// SIMATIC S7-200 project (STEP 7-Micro/WIN), CPU 224 CN REL 02.01

SYMBOL_TABLE 用户定义2
A灯电流             AIW0
B灯电流             AIW2
C灯电流             AIW4
外部机器速度           AIW6
A灯温度             AIW8
B灯温度             AIW10
C灯温度             AIW12
冷水机温度            AIW14
调光变频器频率          AQW0
风机变频器频率          AQW2
急停               I0.0
水流开关             I0.1
变压器A超温           I0.2
变压器B超温           I0.3
变压器C超温           I0.4
A灯限位             I0.5
B灯限位             I0.6
C灯限位             I0.7
A灯快门开启信号         I1.0
B灯快门开启信号         I1.1
C灯快门开启信号         I1.2
长车信号             I1.3
合压信号             I1.4
低水位检测            I1.5
制冷故障             I2.0
风机变频故障           I2.1
冷却系统启动           Q0.0
风机变频启动           Q0.1
A灯启动             Q0.2
B灯启动             Q0.3
C灯启动             Q0.4
A灯开启75           Q0.5
A灯开启100          Q0.6
B灯开启75           Q0.7
B灯开启100          Q1.0
C灯开启75           Q1.1
C灯开启100          Q2.0
A灯快门开启           Q2.1
B灯快门开启           Q2.2
C灯快门开启           Q2.3
报警输出             Q2.4
风机变频复位           Q2.5
风机选择             Q2.6
END_SYMBOL_TABLE

ORGANIZATION_BLOCK 主程序:OB1
TITLE=应用于印刷厂UV固化生产线的PLC控制系统。负责管理照明系统（A灯启动、B灯启动、C灯启动）、冷却系统（冷却系统启动）和通风系统（风机变频启动），确保油墨固化过程在安全、高效的条件下进行。
// 系统通过水流开关和低水位检测监测水况，并在水流正常且水位充足时激活冷却系统启动，为生产线提供稳定的散热支持。
// 冷却系统启动时必须确保水流正常。若冷水机温度超过设定值，系统暂停冷却系统启动并置位报警输出。水流开关检测到异常时，触发报警输出以提示操作员。操作员通过报警复位手动清除报警输出状态，报警复位后应确保报警条件已解除。
// 生产线上的A灯启动、B灯启动、C灯启动分别控制三组UV灯，用于固化不同区域的印刷油墨。这些灯的运行依赖于A灯温度、B灯温度、C灯温度的实时监测，只有在温度低于安全阈值、冷却系统启动和风机变频启动正常运行，且变压器A超温、变压器B超温、变压器C超温未触发时，灯才能开启。A灯启动时，A灯快门保持关闭状态。灯的亮度通过A灯开启75、A灯开启100等输出根据外部机器速度动态调节，确保固化效果与生产节奏匹配。此外，A灯快门开启、B灯快门开启、C灯快门开启在合压信号和长车信号确认生产线处于特定状态时打开，快门开启应在灯启动后特定时间触发。计时器阈值根据生产需求初始化为固定值，存储在系统中。
// 风机变频启动通过风机选择切换模式并在无风机变频故障时启动，为生产线提供通风散热。系统还配备保护机制，例如当A灯限位、B灯限位、C灯限位触发时，激活报警输出并关闭相关灯。急停按钮允许操作员随时中断冷却系统启动等关键输出，确保紧急情况下安全。在实际运行中，系统通过数据处理子程序采集A灯电流、B灯电流、C灯电流和温度数据，调整调光变频器频率和风机变频器频率，优化能耗与性能。生产线运行时间由系统累计记录，并与设定值比较以控制设备状态。当生产线运行时间达到或超过设定值时，停止所有灯。
// 
BEGIN
Network 1 // 网络标题
// 网络注释
LD     SM0.1
R      冷却系统启动:Q0.0, 100
R      M0.0, 100
R      M10.0, 100
R      V1000.0, 26
R      V1003.3, 100
S      M20.0, 1
R      V2700.0, 8
Network 2
LD     M20.0
TON    T45, +300
Network 3
LD     水流开关:I0.1
EU
R      M20.0, 1
Network 4
LD     T45
AN     水流开关:I0.1
S      报警输出:Q2.4, 1
S      V1000.5, 1
Network 5
LD     T45
AN     低水位检测:I1.5
R      A灯启动:Q0.2, 12
S      V1000.6, 1
S      报警输出:Q2.4, 1
R      冷却系统启动:Q0.0, 1
S      M13.7, 1
Network 7
LD     T45
R      M20.0, 1
Network 9
LD     SM0.0
CALL   运行:SBR0
Network 10
LD     SM0.0
CALL   报警:SBR1
Network 11
LD     SM0.0
CALL   数据处理:SBR2
Network 12
LDN    急停:I0.0
R      冷却系统启动:Q0.0, 100
R      M0.0, 100
END_ORGANIZATION_BLOCK

SUBROUTINE_BLOCK 运行:SBR0
TITLE=子程序注释
BEGIN
Network 2
LD     M1.1
EU
AN     制冷故障:I2.0
AW<=   VW806, VW206
A      低水位检测:I1.5
S      冷却系统启动:Q0.0, 1
Network 3
LD     M1.1
ED
R      冷却系统启动:Q0.0, 1
Network 4
LD     M6.0
EU
S      风机选择:Q2.6, 1
Network 5
LD     风机选择:Q2.6
ED
R      M6.0, 1
R      A灯启动:Q0.2, 18
Network 6
LD     冷却系统启动:Q0.0
ED
R      M0.3, 7
R      A灯启动:Q0.2, 18
R      M1.3, 12
Network 7
LD     风机变频启动:Q0.1
ED
R      A灯启动:Q0.2, 18
Network 9
LD     M6.0
ED
R      风机选择:Q2.6, 1
Network 10
LD     M1.2
EU
A      风机选择:Q2.6
AN     风机变频故障:I2.1
S      风机变频启动:Q0.1, 1
Network 11
LD     M1.2
ED
R      风机变频启动:Q0.1, 1
Network 12
LD     M0.3
EU
A      冷却系统启动:Q0.0
A      风机变频启动:Q0.1
AW<=   VW800, VW200
AN     A灯限位:I0.5
AN     V1001.0
A      变压器A超温:I0.2
AN     V1001.1
S      A灯启动:Q0.2, 1
Network 13
LDW>=  VW418, VW2500
A      A灯启动:Q0.2
A      T40
S      A灯开启75:Q0.5, 1
Network 14
LDW<   VW418, VW2600
R      A灯开启75:Q0.5, 1
Network 15
LDW>=  VW418, VW2502
A      A灯启动:Q0.2
A      T40
S      A灯开启100:Q0.6, 1
Network 16
LDW<   VW418, VW2602
R      A灯开启100:Q0.6, 1
Network 17
LD     M0.5
EU
A      冷却系统启动:Q0.0
A      风机变频启动:Q0.1
AW<=   VW802, VW202
AN     B灯限位:I0.6
A      变压器B超温:I0.3
AN     V1001.2
AN     V1001.3
S      B灯启动:Q0.3, 1
Network 18
LDW>=  VW418, VW2504
A      B灯启动:Q0.3
A      T46
S      B灯开启75:Q0.7, 1
Network 19
LDW<   VW418, VW2604
R      B灯开启75:Q0.7, 1
Network 20
LDW>=  VW418, VW2506
A      B灯启动:Q0.3
A      T46
S      B灯开启100:Q1.0, 1
Network 21
LDW<   VW418, VW2606
R      B灯开启100:Q1.0, 1
Network 22
LD     M0.7
EU
A      冷却系统启动:Q0.0
A      风机变频启动:Q0.1
AW<=   VW804, VW204
AN     C灯限位:I0.7
A      变压器C超温:I0.4
AN     V1001.4
AN     V1001.5
S      C灯启动:Q0.4, 1
Network 23
LDW>=  VW418, VW2508
A      C灯启动:Q0.4
A      T47
S      C灯开启75:Q1.1, 1
Network 24
LDW<   VW418, VW2608
R      C灯开启75:Q1.1, 1
Network 25
LDW>=  VW418, VW2510
A      C灯启动:Q0.4
A      T47
S      C灯开启100:Q2.0, 1
Network 26
LDW<   VW418, VW2610
R      C灯开启100:Q2.0, 1
Network 27
LD     M0.4
EU
R      A灯启动:Q0.2, 1
R      A灯开启75:Q0.5, 2
Network 28
LD     M0.6
EU
R      B灯启动:Q0.3, 1
R      B灯开启75:Q0.7, 2
Network 29
LD     M1.0
EU
R      C灯启动:Q0.4, 1
R      C灯开启75:Q1.1, 2
Network 30
LD     合压信号:I1.4
EU
A      长车信号:I1.3
LPS
A      A灯启动:Q0.2
A      T40
AW>=   VW418, VW3000
S      A灯快门开启:Q2.1, 1
LRD
A      B灯启动:Q0.3
A      T46
AW>=   VW418, VW3000
S      B灯快门开启:Q2.2, 1
LPP
A      C灯启动:Q0.4
A      T47
AW>=   VW418, VW3000
S      C灯快门开启:Q2.3, 1
Network 31
LD     T40
EU
A      合压信号:I1.4
A      长车信号:I1.3
A      A灯启动:Q0.2
AW>=   VW418, VW3000
S      A灯快门开启:Q2.1, 1
Network 32
LD     T46
EU
A      合压信号:I1.4
A      长车信号:I1.3
A      B灯启动:Q0.3
AW>=   VW418, VW3000
S      B灯快门开启:Q2.2, 1
Network 33
LD     T47
EU
A      合压信号:I1.4
A      长车信号:I1.3
A      C灯启动:Q0.4
AW>=   VW418, VW3000
S      C灯快门开启:Q2.3, 1
Network 34
LDW>=  VW418, VW3000
EU
A      合压信号:I1.4
A      长车信号:I1.3
LPS
A      A灯启动:Q0.2
A      T40
S      A灯快门开启:Q2.1, 1
LRD
A      B灯启动:Q0.3
A      T46
S      B灯快门开启:Q2.2, 1
LPP
A      C灯启动:Q0.4
A      T47
S      C灯快门开启:Q2.3, 1
Network 35
LDW<   VW418, VW3000
EU
LD     A灯快门开启:Q2.1
O      B灯快门开启:Q2.2
O      C灯快门开启:Q2.3
ALD
R      A灯快门开启:Q2.1, 1
R      B灯快门开启:Q2.2, 1
R      C灯快门开启:Q2.3, 1
Network 46
LD     A灯启动:Q0.2
ED
R      A灯快门开启:Q2.1, 1
Network 47
LD     B灯启动:Q0.3
ED
R      B灯快门开启:Q2.2, 1
Network 48
LD     C灯启动:Q0.4
ED
R      C灯快门开启:Q2.3, 1
Network 51
LD     合压信号:I1.4
ED
A      长车信号:I1.3
LD     A灯快门开启:Q2.1
O      B灯快门开启:Q2.2
O      C灯快门开启:Q2.3
ALD
S      M5.0, 2
Network 52
LD     合压信号:I1.4
EU
A      M5.0
R      M5.0, 1
Network 53
LD     M5.0
TON    T38, VW150
Network 54
LD     T38
EU
R      A灯快门开启:Q2.1, 3
R      M5.0, 1
Network 55
LDN    合压信号:I1.4
A      长车信号:I1.3
LD     A灯启动:Q0.2
O      B灯启动:Q0.3
O      C灯启动:Q0.4
ALD
S      M9.0, 1
Network 56
LDN    合压信号:I1.4
ED
A      长车信号:I1.3
R      M9.0, 1
Network 57
LD     长车信号:I1.3
ED
R      M9.0, 1
Network 58
LD     M9.0
EU
BITIM  VD350
Network 59
LD     M9.0
CITIM  VD350, VD354
Network 60
LD     M9.0
ED
MOVD   +0, VD350
MOVD   +0, VD354
Network 61
LDD>=  VD354, VD304
EU
R      A灯启动:Q0.2, 18
S      报警输出:Q2.4, 1
S      V1000.2, 1
S      M14.1, 1
Network 62
LD     A灯启动:Q0.2
TON    T40, VW2002
Network 63
LD     B灯启动:Q0.3
TON    T46, VW2002
Network 64
LD     C灯启动:Q0.4
TON    T47, VW2002
Network 65
LD     T40
O      T46
O      T47
EU
S      V1003.2, 1
Network 66
LDN    A灯启动:Q0.2
AN     B灯启动:Q0.3
AN     C灯启动:Q0.4
R      V1003.2, 1
Network 69
LD     M7.0
EU
AN     A灯启动:Q0.2
AN     B灯启动:Q0.3
AN     C灯启动:Q0.4
S      A灯快门开启:Q2.1, 1
Network 70
LD     M7.0
ED
AN     A灯启动:Q0.2
AN     B灯启动:Q0.3
AN     C灯启动:Q0.4
R      A灯快门开启:Q2.1, 1
Network 71
LD     M7.1
EU
AN     A灯启动:Q0.2
AN     B灯启动:Q0.3
AN     C灯启动:Q0.4
S      B灯快门开启:Q2.2, 1
Network 72
LD     M7.1
ED
AN     A灯启动:Q0.2
AN     B灯启动:Q0.3
AN     C灯启动:Q0.4
R      B灯快门开启:Q2.2, 1
Network 73
LD     M7.2
EU
AN     A灯启动:Q0.2
AN     B灯启动:Q0.3
AN     C灯启动:Q0.4
S      C灯快门开启:Q2.3, 1
Network 74
LD     M7.2
ED
AN     A灯启动:Q0.2
AN     B灯启动:Q0.3
AN     C灯启动:Q0.4
R      C灯快门开启:Q2.3, 1
Network 75
LDN    A灯开启75:Q0.5
AN     A灯开启100:Q0.6
A      A灯启动:Q0.2
S      Q1.5, 1
Network 76
LD     A灯开启75:Q0.5
O      A灯开启100:Q0.6
R      Q1.5, 1
Network 77
LD     A灯启动:Q0.2
ED
R      Q1.5, 1
R      A灯开启75:Q0.5, 2
Network 78
LDN    B灯开启75:Q0.7
AN     B灯开启100:Q1.0
A      B灯启动:Q0.3
S      Q1.6, 1
Network 79
LD     B灯开启75:Q0.7
O      B灯开启100:Q1.0
R      Q1.6, 1
Network 80
LD     B灯启动:Q0.3
ED
R      Q1.6, 1
R      B灯开启75:Q0.7, 2
Network 82
LDN    C灯开启75:Q1.1
AN     C灯开启100:Q2.0
A      C灯启动:Q0.4
S      Q1.7, 1
Network 83
LD     C灯开启75:Q1.1
O      C灯开启100:Q2.0
R      Q1.7, 1
Network 84
LD     C灯启动:Q0.4
ED
R      Q1.7, 1
R      C灯开启75:Q1.1, 1
R      C灯开启100:Q2.0, 1
END_SUBROUTINE_BLOCK

SUBROUTINE_BLOCK 报警:SBR1
TITLE=
BEGIN
Network 1
LD     M10.0
R      报警输出:Q2.4, 1
R      V1000.3, 100
R      V1000.0, 26
R      M17.0, 4
R      M9.0, 1
Network 2
LDW>   VW520, +120
EU
A      A灯启动:Q0.2
A      T49
S      V2700.0, 1
Network 3
LD     T49
EU
A      A灯启动:Q0.2
AW>    VW520, +120
S      V2700.0, 1
Network 4
LD     V2700.0
TON    T120, 20
Network 5
LD     T120
EU
AW>    VW520, +120
S      V1001.0, 1
S      报警输出:Q2.4, 1
R      A灯启动:Q0.2, 1
R      A灯开启75:Q0.5, 2
R      V2700.0, 1
Network 6
LD     T120
EU
R      V2700.0, 1
Network 7
LDW<   VW520, 40
EU
A      A灯启动:Q0.2
A      T49
S      V2700.1, 1
Network 8
LD     T49
EU
A      A灯启动:Q0.2
AW<    VW520, 40
S      V2700.1, 1
Network 9
LD     V2700.1
TON    T121, 20
Network 10
LD     T121
EU
AW<    VW520, 40
S      V1001.1, 1
S      报警输出:Q2.4, 1
R      A灯启动:Q0.2, 1
R      A灯开启75:Q0.5, 2
R      V2700.1, 1
Network 11
LD     T121
EU
R      V2700.1, 1
Network 14
LD     A灯启动:Q0.2
TON    T49, +300
Network 17
LDW>   VW620, +120
EU
A      B灯启动:Q0.3
A      T50
S      V2700.2, 1
Network 18
LD     T50
EU
AW>    VW620, +120
S      V2700.2, 1
Network 19
LD     V2700.2
TON    T122, 20
Network 20
LD     T122
EU
AW>    VW620, +120
S      V1001.2, 1
S      报警输出:Q2.4, 1
R      B灯启动:Q0.3, 1
R      B灯开启75:Q0.7, 2
R      V2700.2, 1
Network 21
LD     T122
EU
R      V2700.2, 1
Network 23
LD     B灯启动:Q0.3
TON    T50, +300
Network 25
LDW<   VW620, 40
EU
A      B灯启动:Q0.3
A      T50
S      V2700.3, 1
Network 26
LD     T50
EU
A      B灯启动:Q0.3
AW<    VW620, 40
S      V2700.3, 1
Network 27
LD     V2700.3
TON    T123, 20
Network 28
LD     T123
EU
AW<    VW620, 40
S      V1001.3, 1
S      报警输出:Q2.4, 1
R      B灯启动:Q0.3, 1
R      B灯开启75:Q0.7, 2
R      V2700.3, 1
Network 29
LD     T123
EU
R      V2700.3, 1
Network 32
LDW>   VW720, +120
EU
A      C灯启动:Q0.4
A      T51
S      V2700.4, 1
Network 33
LD     T51
EU
A      C灯启动:Q0.4
AW>    VW720, +120
S      V2700.4, 1
Network 34
LD     V2700.4
TON    T124, 20
Network 35
LD     T124
EU
AW>    VW720, +120
S      V1001.4, 1
S      报警输出:Q2.4, 1
R      C灯启动:Q0.4, 1
R      C灯开启75:Q1.1, 2
R      V2700.4, 1
Network 36
LD     T124
EU
R      V2700.4, 1
Network 37
LDW<   VW720, 40
EU
A      C灯启动:Q0.4
A      T51
S      V2700.5, 1
Network 38
LD     T51
EU
A      C灯启动:Q0.4
AW<    VW720, 40
S      V2700.5, 1
Network 39
LD     V2700.5
TON    T125, 20
Network 40
LD     T125
EU
AW<    VW720, 40
S      V1001.5, 1
S      报警输出:Q2.4, 1
R      C灯启动:Q0.4, 1
R      C灯开启75:Q1.1, 2
R      V2700.5, 1
Network 41
LD     T125
EU
R      V2700.5, 1
Network 44
LD     C灯启动:Q0.4
TON    T51, +300
Network 46
LDW>   VW800, VW200
EU
S      M17.0, 1
Network 47
LD     M17.0
TON    T102, 60
Network 48
LD     T102
EU
AW>    VW800, VW200
S      V1001.6, 1
R      A灯启动:Q0.2, 1
S      报警输出:Q2.4, 1
R      A灯开启75:Q0.5, 2
R      M17.0, 1
Network 49
LD     T102
EU
R      M17.0, 1
Network 51
LDW>   VW802, VW202
EU
S      M17.1, 1
Network 52
LD     M17.1
TON    T103, +60
Network 53
LD     T103
EU
AW>    VW802, VW202
S      V1001.7, 1
R      B灯启动:Q0.3, 1
S      报警输出:Q2.4, 1
R      B灯开启75:Q0.7, 2
R      M17.1, 1
Network 54
LD     T103
EU
R      M17.1, 1
Network 57
LDW>   VW804, VW204
EU
S      M17.2, 1
Network 58
LD     M17.2
TON    T104, +60
Network 59
LD     T104
EU
AW>    VW804, VW204
S      V1000.0, 1
R      C灯启动:Q0.4, 1
S      报警输出:Q2.4, 1
R      C灯开启75:Q1.1, 2
R      M17.2, 1
Network 60
LD     T104
EU
R      M17.2, 1
Network 64
LDW>   VW806, VW206
EU
AN     M20.0
S      M17.3, 1
Network 65
LD     M17.3
TON    T105, +60
Network 66
LD     T105
EU
AW>    VW806, VW206
S      V1000.1, 1
R      冷却系统启动:Q0.0, 1
S      报警输出:Q2.4, 1
R      风机变频复位:Q2.5, 2
R      A灯启动:Q0.2, 20
S      M13.0, 1
R      M17.3, 1
Network 67
LD     T105
EU
R      M17.3, 1
Network 70
LD     制冷故障:I2.0
EU
S      M13.1, 1
Network 71
LD     M13.1
TON    T60, +50
Network 72
LD     T60
EU
A      制冷故障:I2.0
R      冷却系统启动:Q0.0, 1
R      A灯启动:Q0.2, 20
R      风机变频复位:Q2.5, 2
S      V1000.3, 1
S      报警输出:Q2.4, 1
R      M13.1, 1
Network 73
LD     T60
AN     制冷故障:I2.0
R      M13.1, 1
Network 75
LDN    变压器A超温:I0.2
EU
R      A灯启动:Q0.2, 1
S      报警输出:Q2.4, 1
S      M13.2, 1
R      A灯开启75:Q0.5, 2
Network 76
LDN    变压器B超温:I0.3
EU
R      B灯启动:Q0.3, 1
S      报警输出:Q2.4, 1
S      M13.3, 1
R      B灯开启75:Q0.7, 2
Network 77
LDN    变压器C超温:I0.4
EU
R      C灯启动:Q0.4, 1
S      报警输出:Q2.4, 1
S      M13.4, 1
R      C灯开启75:Q1.1, 2
Network 79
LD     风机变频故障:I2.1
EU
S      V2700.6, 1
Network 80
LD     V2700.6
TON    T126, 50
Network 81
LD     T126
EU
A      风机变频故障:I2.1
R      风机变频启动:Q0.1, 1
R      A灯启动:Q0.2, 20
R      风机变频复位:Q2.5, 2
S      V1000.4, 1
S      报警输出:Q2.4, 1
S      M13.5, 1
R      V2700.6, 1
Network 82
LD     T126
EU
R      V2700.6, 1
Network 83
LDN    水流开关:I0.1
EU
AN     M20.0
A      冷却系统启动:Q0.0
R      A灯启动:Q0.2, 20
R      风机变频复位:Q2.5, 2
S      V1000.5, 1
S      报警输出:Q2.4, 1
S      M13.6, 1
Network 84
LDN    低水位检测:I1.5
EU
A      冷却系统启动:Q0.0
AN     M20.0
S      V2700.7, 1
Network 85
LD     V2700.7
TON    T127, 50
Network 86
LD     T127
EU
AN     低水位检测:I1.5
R      A灯启动:Q0.2, 20
R      风机变频复位:Q2.5, 2
S      V1000.6, 1
S      报警输出:Q2.4, 1
R      冷却系统启动:Q0.0, 1
S      M13.7, 1
R      V2700.7, 1
Network 87
LD     T127
EU
R      V2700.7, 1
Network 89
LD     A灯快门开启:Q2.1
TON    T41, +50
Network 90
LD     T41
EU
AN     A灯快门开启信号:I1.0
S      V1000.7, 1
R      A灯启动:Q0.2, 1
S      报警输出:Q2.4, 1
R      A灯快门开启:Q2.1, 1
R      A灯开启75:Q0.5, 2
Network 91
LD     B灯快门开启:Q2.2
TON    T42, +50
Network 92
LD     T42
EU
AN     B灯快门开启信号:I1.1
S      V1003.0, 1
R      B灯启动:Q0.3, 1
S      报警输出:Q2.4, 1
R      B灯快门开启:Q2.2, 1
R      B灯开启75:Q0.7, 2
Network 93
LD     C灯快门开启:Q2.3
TON    T43, +50
Network 94
LD     T43
EU
AN     C灯快门开启信号:I1.2
S      V1003.1, 1
R      C灯启动:Q0.4, 1
S      报警输出:Q2.4, 1
R      C灯快门开启:Q2.3, 1
R      C灯开启75:Q1.1, 2
Network 95
LD     A灯限位:I0.5
EU
S      报警输出:Q2.4, 1
R      A灯开启75:Q0.5, 2
R      A灯快门开启:Q2.1, 1
Network 96
LD     B灯限位:I0.6
EU
S      报警输出:Q2.4, 1
R      B灯开启75:Q0.7, 2
R      B灯快门开启:Q2.2, 1
Network 97
LD     C灯限位:I0.7
EU
S      报警输出:Q2.4, 1
R      C灯开启75:Q1.1, 2
R      C灯快门开启:Q2.3, 1
Network 98
LD     A灯快门开启:Q2.1
ED
S      M16.0, 1
Network 99
LD     A灯快门开启:Q2.1
EU
R      M16.0, 1
Network 100
LD     M16.0
TON    T61, +50
Network 101
LD     T61
EU
A      A灯快门开启信号:I1.0
S      V1000.7, 1
R      A灯启动:Q0.2, 1
S      报警输出:Q2.4, 1
R      A灯快门开启:Q2.1, 1
R      A灯开启75:Q0.5, 2
R      M16.0, 1
Network 102
LD     T61
AN     A灯快门开启信号:I1.0
R      M16.0, 1
Network 103
LD     B灯快门开启:Q2.2
ED
S      M16.1, 1
Network 104
LD     B灯快门开启:Q2.2
EU
R      M16.1, 1
Network 105
LD     M16.1
TON    T62, +50
Network 106
LD     T62
EU
A      B灯快门开启信号:I1.1
S      V1003.0, 1
R      B灯启动:Q0.3, 1
S      报警输出:Q2.4, 1
R      B灯快门开启:Q2.2, 1
R      B灯开启75:Q0.7, 2
R      M16.1, 1
Network 107
LD     T62
AN     B灯快门开启信号:I1.1
R      M16.1, 1
Network 109
LD     C灯快门开启:Q2.3
ED
S      M16.2, 1
Network 110
LD     C灯快门开启:Q2.3
EU
R      M16.2, 1
Network 111
LD     M16.2
TON    T63, +50
Network 112
LD     T63
EU
A      C灯快门开启信号:I1.2
S      V1003.1, 1
R      C灯启动:Q0.4, 1
S      报警输出:Q2.4, 1
R      C灯快门开启:Q2.3, 1
R      C灯开启75:Q1.1, 2
R      M16.2, 1
Network 113
LD     T63
AN     C灯快门开启信号:I1.2
R      M16.2, 1
END_SUBROUTINE_BLOCK

SUBROUTINE_BLOCK 数据处理:SBR2
TITLE=
BEGIN
Network 1
LD     SM0.0
MOVW   A灯电流:AIW0, VW500
ITD    VW500, VD504
DTR    VD504, VD508
MOVR   VD508, VD512
*R     0.0040625, VD512
TRUNC  VD512, VD516
DTI    VD516, VW520
Network 2
LD     SM0.0
MOVW   B灯电流:AIW2, VW600
ITD    VW600, VD604
DTR    VD604, VD608
MOVR   VD608, VD612
*R     0.0040625, VD612
TRUNC  VD612, VD616
DTI    VD616, VW620
Network 3
LD     SM0.0
MOVW   C灯电流:AIW4, VW700
ITD    VW700, VD704
DTR    VD704, VD708
MOVR   VD708, VD712
*R     0.0040625, VD712
TRUNC  VD712, VD716
DTI    VD716, VW720
Network 4
LD     SM0.0
MOVW   A灯温度:AIW8, VW800
MOVW   B灯温度:AIW10, VW802
MOVW   C灯温度:AIW12, VW804
MOVW   冷水机温度:AIW14, VW806
Network 5
LD     SM0.0
MOVW   VW208, VW1500
ITD    VW1500, VD1502
DTR    VD1502, VD1506
MOVR   VD1506, VD1510
/R     100.0, VD1510
Network 6
LD     SM0.0
MOVW   VW210, VW1600
ITD    VW1600, VD1602
DTR    VD1602, VD1606
MOVR   VD1606, VD1610
/R     100.0, VD1610
Network 7
LD     SM0.0
MOVW   外部机器速度:AIW6, VW1700
ITD    VW1700, VD1702
DTR    VD1702, VD1706
Network 8
LD     T40
O      T46
O      T47
MOVR   VD1706, VD1800
*R     VD1510, VD1800
TRUNC  VD1800, VD1804
DTI    VD1804, 调光变频器频率:AQW0
Network 9
LD     SM0.0
MOVR   VD1706, VD1850
*R     VD1610, VD1850
TRUNC  VD1850, VD1854
DTI    VD1854, 风机变频器频率:AQW2
Network 10
LD     SM0.0
MOVW   外部机器速度:AIW6, VW400
ITD    VW400, VD402
DTR    VD402, VD406
MOVR   VD406, VD410
*R     0.00625, VD410
TRUNC  VD410, VD414
DTI    VD414, VW418
Network 11
LD     SM0.0
MOVD   VD100, VD300
MOVD   VD300, VD304
*D     +60000, VD304
Network 12
LD     SM0.0
MOVW   VW104, VW2000
MOVW   VW2000, VW2002
*I     +60, VW2002
Network 14
LD     SM0.4
EU
A      A灯启动:Q0.2
+R     1.0, VD4000
+R     1.0, VD4004
Network 15
LD     M11.0
MOVR   0.0, VD4004
Network 16
LD     SM0.0
MOVR   VD4000, VD4010
/R     45.0, VD4010
MOVR   VD4004, VD4022
/R     45.0, VD4022
MOVR   VD4010, VD4014
*R     10.0, VD4014
TRUNC  VD4014, VD4018
MOVR   VD4022, VD4026
*R     10.0, VD4026
TRUNC  VD4026, VD4030
Network 17
LD     SM0.4
EU
A      B灯启动:Q0.3
+R     1.0, VD4040
+R     1.0, VD4044
Network 18
LD     M11.1
MOVR   0.0, VD4044
Network 19
LD     SM0.0
MOVR   VD4040, VD4050
/R     45.0, VD4050
MOVR   VD4044, VD4062
/R     45.0, VD4062
MOVR   VD4050, VD4054
*R     10.0, VD4054
TRUNC  VD4054, VD4058
MOVR   VD4062, VD4066
*R     10.0, VD4066
TRUNC  VD4066, VD4070
Network 20
LD     SM0.4
EU
A      C灯启动:Q0.4
+R     1.0, VD4080
+R     1.0, VD4084
Network 21
LD     M11.2
MOVR   0.0, VD4084
Network 22
LD     SM0.0
MOVR   VD4080, VD4090
/R     45.0, VD4090
MOVR   VD4084, VD4102
/R     45.0, VD4102
MOVR   VD4090, VD4094
*R     10.0, VD4094
TRUNC  VD4094, VD4098
MOVR   VD4102, VD4106
*R     10.0, VD4106
TRUNC  VD4106, VD4120
Network 23
LD     SM0.0
LPS
AW>    VW2500, +10
MOVW   VW2500, VW2600
-I     +10, VW2600
LRD
AW>    VW2502, +10
MOVW   VW2502, VW2602
-I     +10, VW2602
LRD
AW>    VW2504, +10
MOVW   VW2504, VW2604
-I     +10, VW2604
LRD
AW>    VW2506, +10
MOVW   VW2506, VW2606
-I     +10, VW2606
LRD
AW>    VW2508, +10
MOVW   VW2508, VW2608
-I     +10, VW2608
LPP
AW>    VW2510, +10
MOVW   VW2510, VW2610
-I     +10, VW2610
END_SUBROUTINE_BLOCK
